(* IEC 61131-3 sources: CS_4_Aufzugsteuerung/src/Stations/CP112/Steuerung/Class/clsHMI, 1 file *)

(* ---- clsHMI.st ---- *)
(*!
<Class
	Name               = "clsHMI"
	Revision           = "0.0"
	RealtimeTask       = "false"
	CyclicTask         = "true"
	DefCyclictime      = "1 ms"
	BackgroundTask     = "false"
	Sigmatek           = "false"
	OSInterface        = "false"
	HighPriority       = "false"
	Automatic          = "false"
	UpdateMode         = "Prescan"
	SharedCommandTable = "true"
	Objectsize         = "(284,120)">
	<Channels>
		<Server Name="ClassSvr" Visualized="false" Initialize="false" WriteProtected="true" Retentive="false"/>
		<Server Name="sAnf_HMI0" Visualized="true" Initialize="false" WriteProtected="false" Retentive="false"/>
		<Server Name="sAnf_HMI1" Visualized="true" Initialize="false" WriteProtected="false" Retentive="false"/>
		<Server Name="sAnf_HMI2" Visualized="true" Initialize="false" WriteProtected="false" Retentive="false"/>
		<Server Name="sAnf_HMI3" Visualized="true" Initialize="false" WriteProtected="false" Retentive="false"/>
		<Server Name="sAnf_HMIAuf" Visualized="true" Initialize="false" WriteProtected="false" Retentive="false"/>
		<Server Name="sAnf_HMIZu" Visualized="true" Initialize="false" WriteProtected="false" Retentive="false"/>
		<Client Name="cLichtschranke" Required="true" Internal="false"/>
		<Client Name="cTaster1" Required="false" Internal="false"/>
		<Client Name="cTaster2" Required="false" Internal="false"/>
		<Client Name="cTaster3" Required="false" Internal="false"/>
		<Client Name="cTaster4" Required="false" Internal="false"/>
		<Client Name="cTimer1" Required="true" Internal="false"/>
		<Client Name="cTimer2" Required="true" Internal="false"/>
		<Client Name="cTimer3" Required="true" Internal="false"/>
		<Client Name="cTimer4" Required="true" Internal="false"/>
	</Channels>
</Class>
*)
clsHMI : CLASS
  //Servers:
	ClassSvr 	: SvrChCmd_DINT;
	sAnf_HMI0 	: SvrCh_DINT;
	sAnf_HMI1 	: SvrCh_DINT;
	sAnf_HMI2 	: SvrCh_DINT;
	sAnf_HMI3 	: SvrCh_DINT;
	sAnf_HMIAuf 	: SvrCh_DINT;
	sAnf_HMIZu 	: SvrCh_DINT;
  //Clients:
	cTaster1 	: CltCh_DINT;
	cTaster2 	: CltCh_DINT;
	cTaster3 	: CltCh_DINT;
	cTaster4 	: CltCh_DINT;
	cLichtschranke 	: CltCh_DINT;
	cTimer1 	: CltChCmd_clsTimer;
	cTimer2 	: CltChCmd_clsTimer;
	cTimer3 	: CltChCmd_clsTimer;
	cTimer4 	: CltChCmd_clsTimer;
  //Variables:
		xEtage0 	: BOOL;
		xEtage1 	: BOOL;
		xEtage2 	: BOOL;
		xEtage3 	: BOOL;
		xTaster1old 	: DINT;
		xTaster2old 	: DINT;
		xTaster3old 	: DINT;
		xTaster4old 	: DINT;
  //Functions:

	FUNCTION VIRTUAL GLOBAL CyWork
		VAR_INPUT
			EAX 	: UDINT;
		END_VAR
		VAR_OUTPUT
			state (EAX) 	: UDINT;
		END_VAR;

	FUNCTION GLOBAL Etage0
		VAR_OUTPUT
			xOut 	: BOOL;
		END_VAR;

	FUNCTION GLOBAL Etage1
		VAR_OUTPUT
			xOut 	: BOOL;
		END_VAR;

	FUNCTION GLOBAL Etage2
		VAR_OUTPUT
			xOut 	: BOOL;
		END_VAR;

	FUNCTION GLOBAL Etage3
		VAR_OUTPUT
			xOut 	: BOOL;
		END_VAR;

	FUNCTION GLOBAL Tuerzu
		VAR_OUTPUT
			xOut 	: BOOL;
		END_VAR;

	FUNCTION GLOBAL Tuerauf
		VAR_OUTPUT
			xOut 	: BOOL;
		END_VAR;

	FUNCTION GLOBAL Lichtschranke
		VAR_OUTPUT
			xOut 	: DINT;
		END_VAR;
  //Tables:
	FUNCTION @STD
		VAR_OUTPUT
			ret_code	: CONFSTATES;
		END_VAR;
	FUNCTION GLOBAL TAB @CT_;
END_CLASS;

#pragma usingLtd clsTimer

FUNCTION VIRTUAL GLOBAL clsHMI::CyWork
	VAR_INPUT
		EAX : UDINT;
	END_VAR
	VAR_OUTPUT
		state (EAX) : UDINT;
	END_VAR

	// IO lesen
	cTaster1 :=       cTaster1.Read();
	cTaster2 :=       cTaster2.Read();
	cTaster3 :=       cTaster3.Read();
	cTaster4 :=       cTaster4.Read();
  cLichtschranke := cLichtschranke.Read();

	// Etage 0
	IF (cTaster1 <> xTaster1old) OR sAnf_HMI0 THEN
		xTaster1old := cTaster1;
		cTimer1.start(_time := 1000);
	END_IF;

	IF cTimer1.elapsed() THEN
		cTimer1.reset();
	END_IF;

	// Etage 1
	IF (cTaster2 <> xTaster2old) OR sAnf_HMI1 THEN
		xTaster2old := cTaster2;
		cTimer2.start(_time := 1000);
	END_IF;

	IF cTimer2.elapsed() THEN
		cTimer2.reset();
	END_IF;

	// Etage 2
	IF (cTaster3 <> xTaster3old) OR sAnf_HMI2 THEN
		xTaster3old := cTaster3;
		cTimer3.start(_time := 1000);
	END_IF;

	IF cTimer3.elapsed() THEN
		cTimer3.reset();
	END_IF;

	// Etage 3
	IF (cTaster4 <> xTaster4old) OR sAnf_HMI3 THEN
		xTaster4old := cTaster4;
		cTimer4.start(_time := 1000);
	END_IF;

	IF cTimer4.elapsed() THEN
		cTimer4.reset();
	END_IF;

	// Ausgangspulse
	xEtage0 := cTimer1.running();
	xEtage1 := cTimer2.running();
	xEtage2 := cTimer3.running();
	xEtage3 := cTimer4.running();

	state := READY;

END_FUNCTION

FUNCTION GLOBAL clsHMI::Etage0
	VAR_OUTPUT
		xOut 	: BOOL;
	END_VAR
  xOut := xEtage0; //Erkennung falls vom HMI getastet oder vom Schalter
END_FUNCTION

FUNCTION GLOBAL clsHMI::Etage1
	VAR_OUTPUT
		xOut 	: BOOL;
	END_VAR
  xOut := xEtage1; //Erkennung falls vom HMI getastet oder vom Schalter
END_FUNCTION

FUNCTION GLOBAL clsHMI::Etage2
	VAR_OUTPUT
		xOut 	: BOOL;
	END_VAR
  xOut := xEtage2; //Erkennung falls vom HMI getastet oder vom Schalter
END_FUNCTION

FUNCTION GLOBAL clsHMI::Etage3
	VAR_OUTPUT
		xOut 	: BOOL;
	END_VAR
  xOut := xEtage3; //Erkennung falls vom HMI getastet oder vom Schalter
END_FUNCTION

FUNCTION GLOBAL clsHMI::Tuerzu
	VAR_OUTPUT
		xOut 	: BOOL;
	END_VAR
//Erkennung falls vom HMI getastet oder vom Schalter
  IF sAnf_HMIZu > 0 THEN
    xOut := TRUE;
  ELSE
    xOut := FALSE;
  END_IF;
END_FUNCTION

FUNCTION GLOBAL clsHMI::Tuerauf
	VAR_OUTPUT
		xOut 	: BOOL;
	END_VAR
//Erkennung falls vom HMI getastet oder vom Schalter
  IF sAnf_HMIAuf > 0  THEN
    xOut := TRUE;
  ELSE
    xOut := FALSE;
  END_IF;
END_FUNCTION

FUNCTION GLOBAL clsHMI::Lichtschranke
	VAR_OUTPUT
		xOut 	: DINT;
	END_VAR

  xOut :=  cLichtschranke;

END_FUNCTION
